TYPE "MachineState"
VERSION : 0.1
   STRUCT
      running : Bool;
      faulted : Bool;
   END_STRUCT;

END_TYPE

